ABB RobotStudio station: Szymkowiak_Czerwinska_final (1).rspag

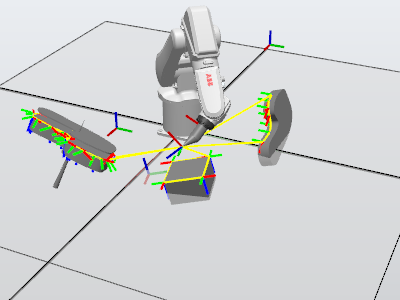
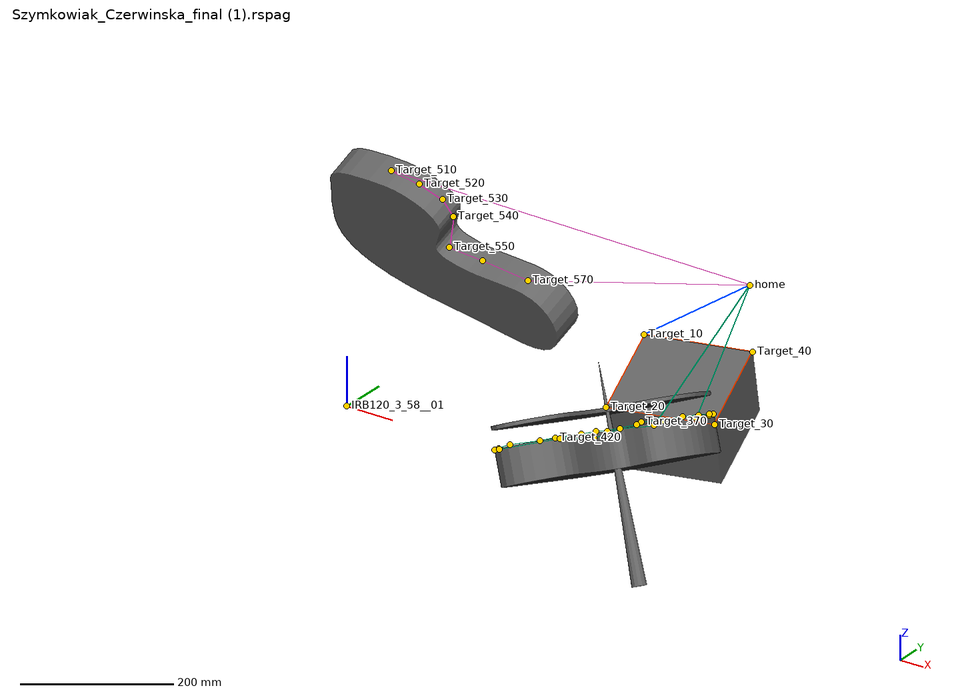
[picture v1: parts stored in the station drawn from their meshes, with robot base, taught points and paths (robot models come from the ABB library and are not in the file)]
--- station ---
Station Station (saved by RobotStudio 25.5.11605.0)
Controller Controller1
  mechanical unit ROB_1: IRB120_3_58__01, 6 joints, base frame (0, 0, 0) mm
Layout (positions relative to the parent item):
  - IRB120_3_58__01 [mechanism, from %ABB.RobotStudio.Models.IRB120%\IRB120_3_58_G_01.rslib] at (0, 0, 0) mm; joint values [0.7069, 0.7737, 0.0512, -1.3169, 0.7984, 0.0181] (rad or m)
  - Gwozdz [mechanism] at (389.5, 267.05, 263.13) mm, rotated rx -133.7 ry -23.28 rz -92.59 deg
      TCP Gwozdz at (13.78, -22.95, 107.1) mm, rotated rx 22.5 ry 12.3 rz 0 deg
      links: Group_1
  - Part_4 [part] at (356.82, 20.61, -19.41) mm, rotated rx 15 ry 0 rz 15 deg, size 150 x 150 x 100 mm
  - spline [graphiccomponentgroup] at (842.54, 100.2, 183.59) mm, rotated rx 23.86 ry -17.62 rz -89.19 deg
    - Part_8 [part], size 356.2 x 175.5 x 50 mm
    - Part_10 [part] at (47.75, 249.87, 75.62) mm, size 356.2 x 175.5 x 5 mm
    - Part_5 [part] at (-233.39, -133.39, -154.61) mm, size 20 x 20 x 300 mm
  - 3 [graphiccomponentgroup] at (660.88, 255.89, -87.62) mm
    - Part_6 [part] at (-929.3, 12.05, 504.16) mm, rotated rx 110.54 ry 15.88 rz 5.85 deg, size 356.2 x 175.5 x 50 mm
Attachment: Gwozdz is attached to IRB120_3_58__01 / Link6
Attachment: Workobject_A is attached to Part_4
Attachment: Spline_2 is attached to spline
Attachment: gitara is attached to Part_6
Collision set CollisionSet_1: Gwozdz, IRB120_3_58__01 against Part_4, near miss 0 m
Collision set CollisionSet_2: Gwozdz, IRB120_3_58__01 against spline, near miss 0 m
Collision set CollisionSet_3: Gwozdz, IRB120_3_58__01 against 3, near miss 0 m

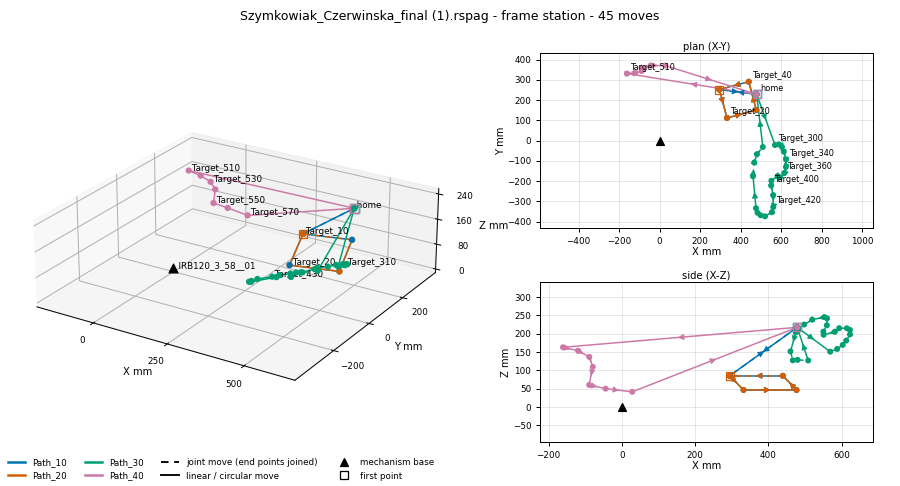
[picture p0: tool path of Szymkowiak_Czerwinska_final (1).rspag in frame station, 45 of 45 moves have a stored position in this frame; points joined in program order, loops and branches not executed]
--- Backups/Controller1/RAPID/TASK1/PROGMOD/CalibData.mod ---
MODULE CalibData
    PERS tooldata Gwozdz:=[TRUE,[[13.78,-22.949,104.2],[0.975140697,0.193967545,0.105073248,-0.020900368]],[1,[0,0,1],[1,0,0,0],0,0,0]];
    TASK PERS wobjdata Workobject_A:=[FALSE,TRUE,"",[[356.824039201,20.610713144,-19.411428383],[0.982962913,0.129409523,0.017037087,0.129409523]],[[0,0,0],[1,0,0,0]]];
    TASK PERS wobjdata Workobject_3:=[FALSE,TRUE,"",[[90.527,-395.87,5.743],[1,0,0,0]],[[0,0,0],[1,0,0,0]]];
    TASK PERS wobjdata Spline_2:=[FALSE,TRUE,"",[[189.277,-219.99,50],[1,0,0,0]],[[0,0,0],[1,0,0,0]]];
    TASK PERS wobjdata gitara:=[FALSE,TRUE,"",[[-733.881,111.122,140.989],[1,0,0,0]],[[0,0,0],[1,0,0,0]]];
ENDMODULE

--- Backups/Controller1/RAPID/TASK1/PROGMOD/Module1.mod ---
MODULE Module1
    CONST robtarget Target_10:=[[-0.000115513,258.709411951,39.203781036],[0,-0.70710678,0.707106782,0],[0,0,-2,0],[9E+09,9E+09,9E+09,9E+09,9E+09,9E+09]];
    CONST robtarget Target_20:=[[-0.000115649,108.709411951,39.203781178],[0,-0.70710678,0.707106782,0],[0,0,-2,0],[9E+09,9E+09,9E+09,9E+09,9E+09,9E+09]];
    CONST robtarget Target_30:=[[149.99988435,108.709411815,39.203781214],[0,1,0,0],[0,-1,-2,0],[9E+09,9E+09,9E+09,9E+09,9E+09,9E+09]];
    CONST robtarget Target_40:=[[149.999884487,258.709411815,39.203781073],[0,0.707106782,0.70710678,0],[0,-1,-3,0],[9E+09,9E+09,9E+09,9E+09,9E+09,9E+09]];
    CONST robtarget Target_50:=[[-0.000115513,258.709411951,39.203781036],[0,0,1,0],[0,0,0,0],[9E+09,9E+09,9E+09,9E+09,9E+09,9E+09]];
    CONST robtarget Target_60:=[[32.293288585,-26.274,94.875020901],[0.343932459,0.492118694,0.617827212,0.507758989],[-2,0,-1,0],[9E+09,9E+09,9E+09,9E+09,9E+09,9E+09]];
    CONST robtarget Target_70:=[[25.747933082,1.085485712,96.628843622],[0.39672232,0.534698929,0.585330164,0.46270623],[-2,0,-1,0],[9E+09,9E+09,9E+09,9E+09,9E+09,9E+09]];
    CONST robtarget Target_80:=[[26.021259984,11.796174998,96.555605899],[0.494711421,0.608618518,0.505233223,0.359977081],[-2,1,-2,0],[9E+09,9E+09,9E+09,9E+09,9E+09,9E+09]];
    CONST robtarget Target_90:=[[30.549792469,18.944,95.342189277],[0.643544046,0.697450705,0.293003516,0.116458208],[0,0,0,0],[9E+09,9E+09,9E+09,9E+09,9E+09,9E+09]];
    CONST robtarget Target_100:=[[41.243529195,21.890992963,92.476811157],[0.698217822,0.703354067,0.111767046,-0.072753394],[0,0,0,0],[9E+09,9E+09,9E+09,9E+09,9E+09,9E+09]];
    CONST robtarget Target_110:=[[54.698904052,21.13,88.87145433],[0.705708942,0.69316434,0.044439723,-0.139725438],[0,0,0,0],[9E+09,9E+09,9E+09,9E+09,9E+09,9E+09]];
    CONST robtarget Target_120:=[[84.871273532,12.465734711,80.786792294],[0.705846315,0.670872595,-0.04220165,-0.223450133],[0,0,0,0],[9E+09,9E+09,9E+09,9E+09,9E+09,9E+09]];
    CONST robtarget Target_130:=[[112.133819609,0.297,73.481815089],[0.705711324,0.670172739,-0.044401889,-0.225540462],[0,0,0,0],[9E+09,9E+09,9E+09,9E+09,9E+09,9E+09]];
    CONST robtarget Target_140:=[[181.80121983,-27.286,54.814491461],[0.702817485,0.658742185,-0.077766204,-0.257018935],[0,0,0,0],[9E+09,9E+09,9E+09,9E+09,9E+09,9E+09]];
    CONST robtarget Target_150:=[[203.084989416,-41.869542951,49.111522589],[0.691191833,0.62903013,-0.149177244,-0.322987763],[0,0,0,0],[9E+09,9E+09,9E+09,9E+09,9E+09,9E+09]];
    CONST robtarget Target_160:=[[221.549955545,-60.687523743,44.163849826],[0.676034315,0.599343122,-0.207310409,-0.375217033],[0,0,0,0],[9E+09,9E+09,9E+09,9E+09,9E+09,9E+09]];
    CONST robtarget Target_170:=[[238.959203727,-84.186992664,39.499055835],[0.664110287,0.578636982,-0.242811712,-0.406422493],[0,0,0,0],[9E+09,9E+09,9E+09,9E+09,9E+09,9E+09]];
    CONST robtarget Target_180:=[[257.075819472,-112.815,34.644723277],[0.65833708,0.569115287,-0.258054817,-0.419651987],[0,0,0,0],[9E+09,9E+09,9E+09,9E+09,9E+09,9E+09]];
    CONST robtarget Target_190:=[[298.990897184,-186.304854501,23.413612053],[0.650010389,0.555815927,-0.278363961,-0.437114007],[0,0,0,0],[9E+09,9E+09,9E+09,9E+09,9E+09,9E+09]];
    CONST robtarget Target_200:=[[318.524416429,-225.602978625,18.179621346],[0.642387659,0.544009988,-0.295530193,-0.451722407],[0,0,0,0],[9E+09,9E+09,9E+09,9E+09,9E+09,9E+09]];
    CONST robtarget Target_210:=[[334.227468572,-263.176581732,13.972001206],[0.629116005,0.524127313,-0.322820464,-0.474647827],[0,0,0,0],[9E+09,9E+09,9E+09,9E+09,9E+09,9E+09]];
    CONST robtarget Target_220:=[[343.939213089,-296.455674623,11.369747105],[0.601571426,0.484887423,-0.371633986,-0.514669007],[0,0,0,0],[9E+09,9E+09,9E+09,9E+09,9E+09,9E+09]];
    CONST robtarget Target_230:=[[345.498809459,-322.870268097,10.951854517],[0.527081739,0.387123658,-0.47136487,-0.591722294],[0,0,0,0],[9E+09,9E+09,9E+09,9E+09,9E+09,9E+09]];
    CONST robtarget Target_240:=[[336.745417159,-339.850372956,13.297318915],[0.30987709,0.134815174,-0.635591212,-0.694136059],[0,0,0,0],[9E+09,9E+09,9E+09,9E+09,9E+09,9E+09]];
    CONST robtarget Target_250:=[[327.826087594,-343.99937053,15.687246069],[0.171520784,-0.011870608,-0.68598879,-0.707007135],[0,0,0,0],[9E+09,9E+09,9E+09,9E+09,9E+09,9E+09]];
    CONST robtarget Target_260:=[[315.518195666,-344.826,18.985135772],[0.069659143,-0.114836922,-0.703667254,-0.697719486],[0,0,0,0],[9E+09,9E+09,9E+09,9E+09,9E+09,9E+09]];
    CONST robtarget Target_270:=[[296.741306529,-342.504994924,24.016388052],[0.058243886,-0.126131528,-0.704703945,-0.695766367],[0,0,0,0],[9E+09,9E+09,9E+09,9E+09,9E+09,9E+09]];
    CONST robtarget Target_280:=[[280.016557847,-344.15,28.497770955],[0.250015953,0.07030572,-0.661431798,-0.703602946],[0,0,0,0],[9E+09,9E+09,9E+09,9E+09,9E+09,9E+09]];
    CONST robtarget Target_290:=[[273.743639455,-350.366155686,30.178594373],[0.42375383,0.262805656,-0.566067744,-0.656455015],[0,0,0,0],[9E+09,9E+09,9E+09,9E+09,9E+09,9E+09]];
    CONST robtarget Target_300:=[[379.818187376,198.530285249,101.14340374],[0.080794632,-0.064061007,0.870872366,-0.480572301],[0,-1,0,0],[9E+09,9E+09,9E+09,9E+09,9E+09,9E+09]];
    CONST robtarget Target_310:=[[398.798930616,201.55355769,108.644212296],[0.005997032,-0.052439583,0.797191505,-0.601414857],[0,-1,0,0],[9E+09,9E+09,9E+09,9E+09,9E+09,9E+09]];
    CONST robtarget Target_320:=[[414.060612159,189.159616563,119.648393506],[0.15313745,0.408655647,0.866532524,-0.242220703],[0,-1,0,0],[9E+09,9E+09,9E+09,9E+09,9E+09,9E+09]];
    CONST robtarget Target_330:=[[423.577274376,165.647663464,131.419216891],[0.196962097,0.54712541,0.74590824,-0.324777794],[0,-1,1,0],[9E+09,9E+09,9E+09,9E+09,9E+09,9E+09]];
    CONST robtarget Target_340:=[[434.035311555,127.327516374,148.236680199],[0.204407328,0.758318384,0.60417945,-0.134677633],[0,-1,1,0],[9E+09,9E+09,9E+09,9E+09,9E+09,9E+09]];
    CONST robtarget Target_350:=[[433.75156002,90.454896969,160.504946511],[0.126225144,0.642321975,0.742941887,-0.139739207],[-1,-1,0,0],[9E+09,9E+09,9E+09,9E+09,9E+09,9E+09]];
    CONST robtarget Target_360:=[[425.32521943,59.992973584,165.098796736],[0.061967959,0.82800912,0.555316016,0.046743884],[-1,-1,1,0],[9E+09,9E+09,9E+09,9E+09,9E+09,9E+09]];
    CONST robtarget Target_370:=[[404.422989752,38.703354806,165.406282644],[0.132456897,-0.907467112,-0.022002682,-0.398088549],[-1,0,1,0],[9E+09,9E+09,9E+09,9E+09,9E+09,9E+09]];
    CONST robtarget Target_380:=[[392.69942564,45.287768591,155.735730099],[0.034407024,-0.851655969,-0.466716338,-0.235953655],[-1,0,1,0],[9E+09,9E+09,9E+09,9E+09,9E+09,9E+09]];
    CONST robtarget Target_390:=[[361.911361181,22.375329586,147.092090309],[0.132921404,0.826414064,0.542391472,-0.071994346],[-1,-1,1,0],[9E+09,9E+09,9E+09,9E+09,9E+09,9E+09]];
    CONST robtarget Target_400:=[[361.144638736,-1.215988604,155.914989553],[0.120961235,0.84291138,0.521875598,-0.050146234],[-1,-1,1,0],[9E+09,9E+09,9E+09,9E+09,9E+09,9E+09]];
    CONST robtarget Target_410:=[[370.709808372,-48.157952098,173.271661643],[0.097142097,0.829595447,0.545283587,-0.070715041],[-1,-1,1,0],[9E+09,9E+09,9E+09,9E+09,9E+09,9E+09]];
    CONST robtarget Target_420:=[[371.21341414,-107.65967769,192.159086411],[0.142548065,0.564425354,0.778671638,-0.234039632],[-1,-1,0,0],[9E+09,9E+09,9E+09,9E+09,9E+09,9E+09]];
    CONST robtarget home:=[[479.039020595,228.419373597,217.688268521],[0.189358781,-0.606844127,0.502209167,-0.586233239],[0,-1,0,0],[9E+09,9E+09,9E+09,9E+09,9E+09,9E+09]];
    CONST robtarget Target_430:=[[364.347539311,-132.881202283,195.549228134],[0.131223185,0.799918218,0.585270789,-0.01922039],[-1,-1,0,0],[9E+09,9E+09,9E+09,9E+09,9E+09,9E+09]];
    CONST robtarget Target_440:=[[330.671113835,-153.291694033,188.62816963],[0.065409955,0.881565205,0.219488312,0.412782278],[-1,0,0,0],[9E+09,9E+09,9E+09,9E+09,9E+09,9E+09]];
    CONST robtarget Target_450:=[[308.873092537,-147.99782022,175.23553106],[0.002837859,0.929421061,0.299920175,0.214979831],[-1,0,1,0],[9E+09,9E+09,9E+09,9E+09,9E+09,9E+09]];
    CONST robtarget Target_460:=[[293.509097881,-135.339550632,164.101209237],[0.148194352,-0.93312273,0.206182801,-0.254576231],[-1,0,1,0],[9E+09,9E+09,9E+09,9E+09,9E+09,9E+09]];
    CONST robtarget Target_470:=[[286.005473037,-113.036967666,153.649542348],[0.119156571,-0.830173017,0.329649022,-0.433527389],[-1,0,1,0],[9E+09,9E+09,9E+09,9E+09,9E+09,9E+09]];
    CONST robtarget Target_480:=[[271.326760585,44.643984375,101.96446254],[0.235016198,-0.577377657,0.633042861,-0.458976213],[-1,1,1,0],[9E+09,9E+09,9E+09,9E+09,9E+09,9E+09]];
    CONST robtarget Target_490:=[[277.736043143,112.556253411,77.54974934],[0.224942367,-0.742618228,0.488872356,-0.398651375],[-1,1,1,0],[9E+09,9E+09,9E+09,9E+09,9E+09,9E+09]];
    CONST robtarget Target_500:=[[325.559577911,183.522556178,74.273225749],[0.15927241,-0.178140553,0.907828431,-0.3445951],[0,-1,4,0],[9E+09,9E+09,9E+09,9E+09,9E+09,9E+09]];
    CONST robtarget Target_520:=[[614.214194066,223.582,12.938004228],[0,0.939692621,0,-0.342020143],[0,0,-2,0],[9E+09,9E+09,9E+09,9E+09,9E+09,9E+09]];
    CONST robtarget Target_530:=[[644.969447518,232.344,-4.131767247],[0,0.939692621,0,-0.342020143],[0,0,-2,0],[9E+09,9E+09,9E+09,9E+09,9E+09,9E+09]];
    CONST robtarget Target_495:=[[299.935371666,166.502951861,72.039805608],[0.187827929,-0.667412492,0.62384148,-0.360697992],[-1,0,2,0],[9E+09,9E+09,9E+09,9E+09,9E+09,9E+09]];
    CONST robtarget Target_510:=[[573.029582644,219.866,22.166500105],[0,0.939692621,0,-0.342020143],[1,0,-2,0],[9E+09,9E+09,9E+09,9E+09,9E+09,9E+09]];
    CONST robtarget Target_540:=[[654.605500324,243.683,-31.22121015],[0,0.939692621,0,-0.342020143],[0,0,-2,0],[9E+09,9E+09,9E+09,9E+09,9E+09,9E+09]];
    CONST robtarget Target_550:=[[644.521305062,248.916,-80.6473513],[0,0.939692621,0,-0.342020143],[0,0,-2,0],[9E+09,9E+09,9E+09,9E+09,9E+09,9E+09]];
    CONST robtarget Target_560:=[[689.496774347,259.629,-90.892520304],[0,0.939692621,0,-0.342020143],[0,0,-2,0],[9E+09,9E+09,9E+09,9E+09,9E+09,9E+09]];
    CONST robtarget Target_570:=[[762.138368671,259.345,-99.429023647],[0,0.939692621,0,-0.342020143],[0,0,-2,0],[9E+09,9E+09,9E+09,9E+09,9E+09,9E+09]];
    CONST robtarget Target_580:=[[734.655,267.963,-95.69],[0.202644877,0,-0.979252293,0],[0,1,-1,0],[9E+09,9E+09,9E+09,9E+09,9E+09,9E+09]];
    CONST robtarget Target_590:=[[290.719680498,153.490427714,78.778602288],[0.292789453,-0.718578623,0.449827742,-0.442237608],[-1,1,1,0],[9E+09,9E+09,9E+09,9E+09,9E+09,9E+09]];
    CONST robtarget Target_600:=[[319.748354811,188.814701144,77.069595791],[0.189358802,-0.606844041,0.502209025,-0.586233442],[0,-2,0,0],[9E+09,9E+09,9E+09,9E+09,9E+09,9E+09]];

    PROC main()
        Path_10;
        Path_30;
        Path_40;
    ENDPROC

    PROC Path_10()
        MoveL home,v1000,fine,Gwozdz\WObj:=wobj0;
        MoveJ Target_10,v50,fine,Gwozdz\WObj:=Workobject_A;
        MoveL Target_20,v50,fine,Gwozdz\WObj:=Workobject_A;
        MoveL Target_30,v50,fine,Gwozdz\WObj:=Workobject_A;
        MoveL Target_40,v50,fine,Gwozdz\WObj:=Workobject_A;
        MoveL Target_50,v50,fine,Gwozdz\WObj:=Workobject_A;
        MoveL home,v1000,fine,Gwozdz\WObj:=wobj0;
    ENDPROC

    PROC Path_20()
        MoveJ Target_10,v1000,fine,Gwozdz\WObj:=Workobject_A;
        MoveL Target_20,v1000,fine,Gwozdz\WObj:=Workobject_A;
        MoveL Target_30,v1000,fine,Gwozdz\WObj:=Workobject_A;
        MoveL Target_40,v1000,fine,Gwozdz\WObj:=Workobject_A;
        MoveJ Target_50,v1000,fine,Gwozdz\WObj:=Workobject_A;
    ENDPROC
    PROC Path_30()
        MoveL home,v1000,fine,Gwozdz\WObj:=wobj0;
        MoveL Target_300,v30,fine,Gwozdz\WObj:=Spline_2;
        MoveL Target_310,v30,fine,Gwozdz\WObj:=Spline_2;
        MoveL Target_320,v30,fine,Gwozdz\WObj:=Spline_2;
        MoveL Target_330,v30,fine,Gwozdz\WObj:=Spline_2;
        MoveL Target_340,v30,fine,Gwozdz\WObj:=Spline_2;
        MoveL Target_350,v30,fine,Gwozdz\WObj:=Spline_2;
        MoveL Target_360,v30,fine,Gwozdz\WObj:=Spline_2;
        MoveL Target_370,v30,fine,Gwozdz\WObj:=Spline_2;
        MoveL Target_380,v30,fine,Gwozdz\WObj:=Spline_2;
        MoveL Target_390,v30,fine,Gwozdz\WObj:=Spline_2;
        MoveL Target_400,v30,fine,Gwozdz\WObj:=Spline_2;
        MoveL Target_410,v30,fine,Gwozdz\WObj:=Spline_2;
        MoveL Target_420,v30,fine,Gwozdz\WObj:=Spline_2;
        MoveL Target_430,v30,fine,Gwozdz\WObj:=Spline_2;
        MoveL Target_440,v30,fine,Gwozdz\WObj:=Spline_2;
        MoveL Target_450,v30,fine,Gwozdz\WObj:=Spline_2;
        MoveL Target_460,v30,fine,Gwozdz\WObj:=Spline_2;
        MoveL Target_470,v30,fine,Gwozdz\WObj:=Spline_2;
        MoveL Target_480,v30,fine,Gwozdz\WObj:=Spline_2;
        MoveJ Target_490,v30,fine,Gwozdz\WObj:=Spline_2;
        MoveJ Target_590,v1000,fine,Gwozdz\WObj:=Spline_2;
        MoveJ Target_600,v1000,fine,Gwozdz\WObj:=Spline_2;
        MoveL home,v1000,fine,Gwozdz\WObj:=wobj0;
    ENDPROC
    PROC Path_40()
        MoveL home,v1000,fine,Gwozdz\WObj:=wobj0;
        MoveL Target_510,v20,fine,Gwozdz\WObj:=gitara;
        MoveL Target_520,v20,fine,Gwozdz\WObj:=gitara;
        MoveL Target_530,v20,z100,Gwozdz\WObj:=gitara;
        MoveL Target_540,v20,z100,Gwozdz\WObj:=gitara;
        MoveL Target_550,v20,z100,Gwozdz\WObj:=gitara;
        MoveL Target_560,v20,fine,Gwozdz\WObj:=gitara;
        MoveL Target_570,v20,fine,Gwozdz\WObj:=gitara;
        MoveL home,v1000,fine,Gwozdz\WObj:=wobj0;
    ENDPROC
ENDMODULE
